// TIA Portal V20 export
ORGANIZATION_BLOCK "CyclicInterrupt"   // OB35, LAD, CyclicInterrupt
{ S7_Optimized_Access := 'TRUE' }
// stored: AutoNumber false, SetENOAutomatically true
BEGIN
END_ORGANIZATION_BLOCK
